TYPE MDP5001_341_7CD731EE :
STRUCT
	MDP5001_341_Input	: MDP5001_341_I_7CD731EE;
	MDP5001_341_Output	: MDP5001_341_O_7CD731EE;
END_STRUCT
END_TYPE

(* stored: Version 1.1.0.1, ProductVersion 3.1.4024.12
   DUT MDP5001_341_7CD731EE: Id {b2a228ca-de0c-4097-9290-a49b3a1e02be} *)
